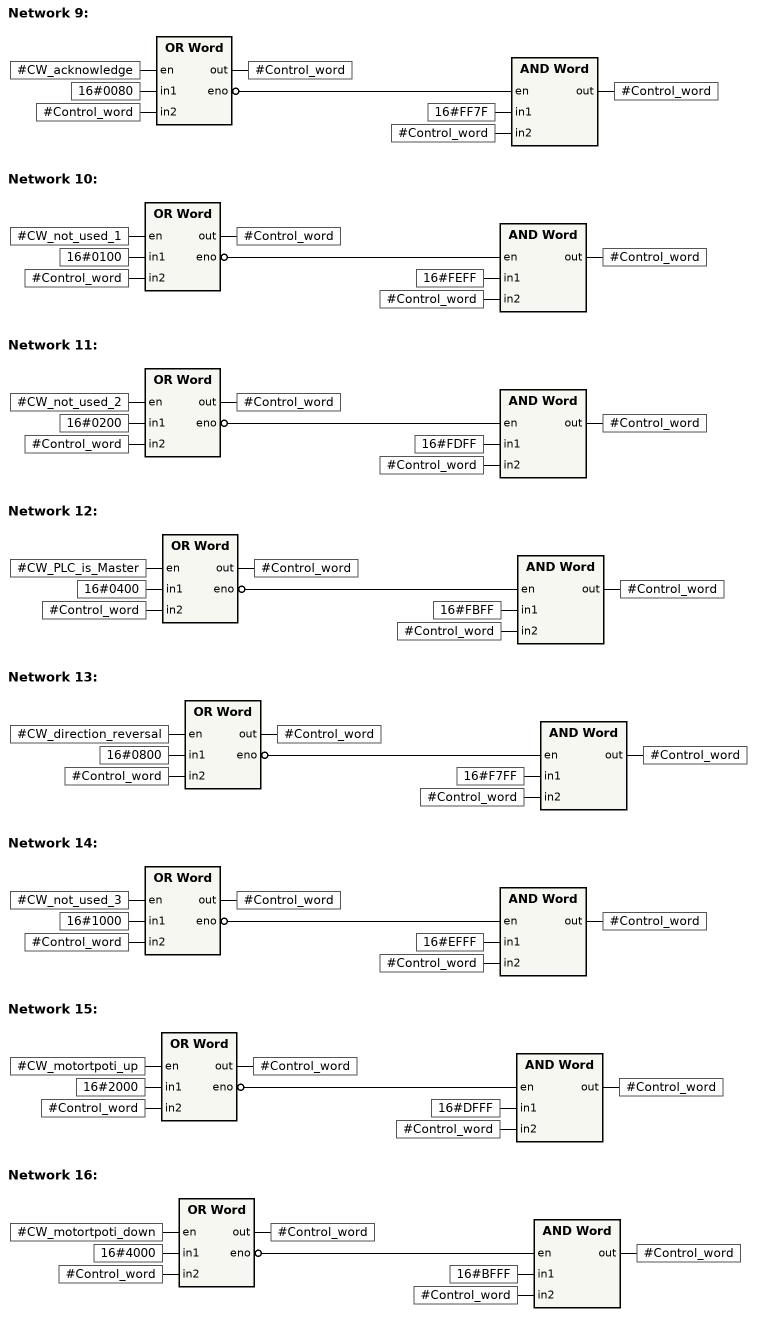
   IF #CW_acknowledge THEN #Control_word := 16#0080 OR #Control_word; END_IF;
   IF NOT #CW_acknowledge THEN #Control_word := 16#FF7F AND #Control_word; END_IF;
END_REGION

REGION Network 10
   IF #CW_not_used_1 THEN #Control_word := 16#0100 OR #Control_word; END_IF;
   IF NOT #CW_not_used_1 THEN #Control_word := 16#FEFF AND #Control_word; END_IF;
END_REGION

REGION Network 11
   IF #CW_not_used_2 THEN #Control_word := 16#0200 OR #Control_word; END_IF;
   IF NOT #CW_not_used_2 THEN #Control_word := 16#FDFF AND #Control_word; END_IF;
END_REGION

REGION Network 12
   IF #CW_PLC_is_Master THEN #Control_word := 16#0400 OR #Control_word; END_IF;
   IF NOT #CW_PLC_is_Master THEN #Control_word := 16#FBFF AND #Control_word; END_IF;
END_REGION

REGION Network 13
   IF #CW_direction_reversal THEN #Control_word := 16#0800 OR #Control_word; END_IF;
   IF NOT #CW_direction_reversal THEN #Control_word := 16#F7FF AND #Control_word; END_IF;
END_REGION

REGION Network 14
   IF #CW_not_used_3 THEN #Control_word := 16#1000 OR #Control_word; END_IF;
   IF NOT #CW_not_used_3 THEN #Control_word := 16#EFFF AND #Control_word; END_IF;
END_REGION

REGION Network 15
   IF #CW_motortpoti_up THEN #Control_word := 16#2000 OR #Control_word; END_IF;
   IF NOT #CW_motortpoti_up THEN #Control_word := 16#DFFF AND #Control_word; END_IF;
END_REGION

REGION Network 16
   IF #CW_motortpoti_down THEN #Control_word := 16#4000 OR #Control_word; END_IF;
   IF NOT #CW_motortpoti_down THEN #Control_word := 16#BFFF AND #Control_word; END_IF;
END_REGION

REGION Network 17
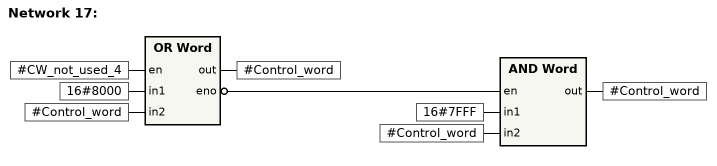
   IF #CW_not_used_4 THEN #Control_word := 16#8000 OR #Control_word; END_IF;
   IF NOT #CW_not_used_4 THEN #Control_word := 16#7FFF AND #Control_word; END_IF;
END_REGION
END_FUNCTION

FUNCTION_BLOCK "Inverter_Process_Data"   // FB1, FBD
{ S7_Optimized_Access := 'TRUE' }
VERSION : 0.1
// stored: AutoNumber false, IsIECCheckEnabled false, IsRetainMemResEnabled false, MemoryReserve 100, SetENOAutomatically false, UDAEnableTagReadback false
   VAR_INPUT
      control_word : Word := 16#0000;
      setpoint : Real;
      RD_address : HW_SUBMODULE;
      WR_address : HW_SUBMODULE;
      ref_quantity : Struct
         speed_p2000 : Real := 1500.0;
         current_p2002 : Real := 0.65;
         torque_p2003 : Real := 1.7;
      END_STRUCT;
   END_VAR
   VAR_OUTPUT
      status_word : Word;
      actual_speed : Real;
      actual_current : Real;
      actual_torque : Real;
      actual_alarm : Word;
      actual_fault : Word;
      RETVAL_RD : Word;
      RETVAL_WR : Word;
   END_VAR
   VAR_TEMP
      InData : Array[1..6] of Word;
      OutData : Array[1..6] of Word;
      actual_speed_INT : Int;
      actual_current_INT : Int;
      actual_torque_INT : Int;
      setpoint_INT : Int;
   END_VAR
BEGIN

REGION Network 1
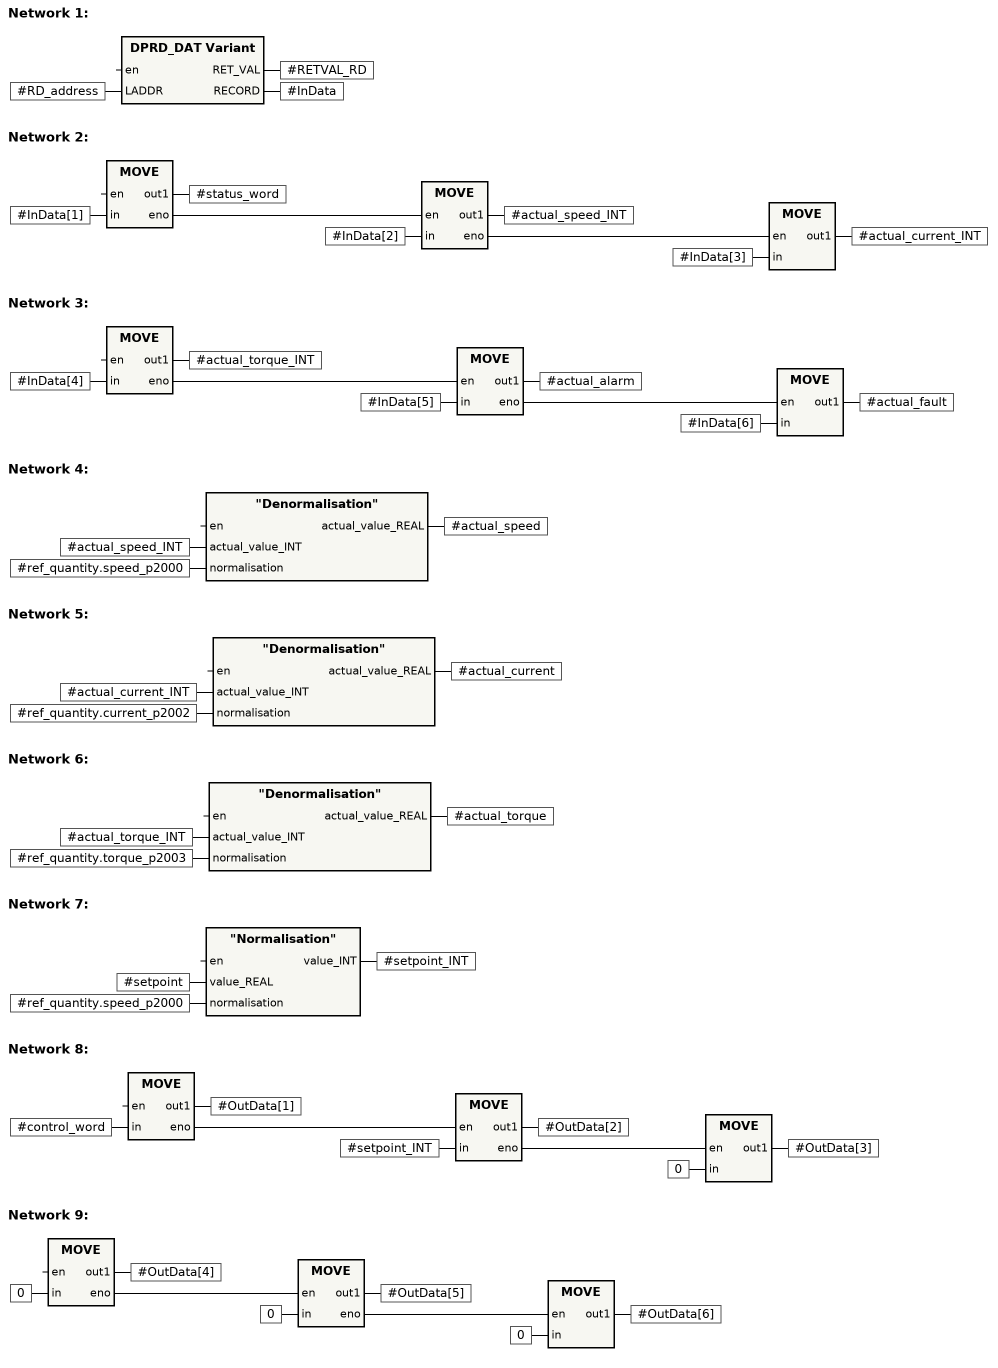
   #RETVAL_RD := DPRD_DAT(LADDR := #RD_address, RECORD => #InData);
END_REGION

REGION Network 2
   // ENO of a box is taken as its EN; it also drops when the box reports an error
   #status_word := #InData[1];
   #actual_speed_INT := #InData[2];
   #actual_current_INT := #InData[3];
END_REGION

REGION Network 3
   // ENO of a box is taken as its EN; it also drops when the box reports an error
   #actual_torque_INT := #InData[4];
   #actual_alarm := #InData[5];
   #actual_fault := #InData[6];
END_REGION

REGION Network 4
   "Denormalisation"(actual_value_INT := #actual_speed_INT,
                     normalisation := #ref_quantity.speed_p2000,
                     actual_value_REAL => #actual_speed);
END_REGION

REGION Network 5
   "Denormalisation"(actual_value_INT := #actual_current_INT,
                     normalisation := #ref_quantity.current_p2002,
                     actual_value_REAL => #actual_current);
END_REGION

REGION Network 6
   "Denormalisation"(actual_value_INT := #actual_torque_INT,
                     normalisation := #ref_quantity.torque_p2003,
                     actual_value_REAL => #actual_torque);
END_REGION

REGION Network 7
   "Normalisation"(value_REAL := #setpoint,
                   normalisation := #ref_quantity.speed_p2000,
                   value_INT => #setpoint_INT);
END_REGION

REGION Network 8
   // ENO of a box is taken as its EN; it also drops when the box reports an error
   #OutData[1] := #control_word;
   #OutData[2] := #setpoint_INT;
   #OutData[3] := 0;
END_REGION

REGION Network 9
   // ENO of a box is taken as its EN; it also drops when the box reports an error
   #OutData[4] := 0;
   #OutData[5] := 0;
   #OutData[6] := 0;
END_REGION

REGION Network 10
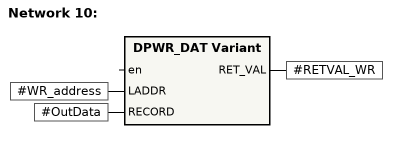
   #RETVAL_WR := DPWR_DAT(LADDR := #WR_address, RECORD := #OutData);
END_REGION
END_FUNCTION_BLOCK

FUNCTION_BLOCK "Modbus"   // FB20, FBD
{ S7_Optimized_Access := 'FALSE' }
VERSION : 0.1
// stored: AutoNumber false, IsIECCheckEnabled false, SetENOAutomatically false, UDAEnableTagReadback false
   VAR_INPUT
      BAUDRATE : UDInt := 115200;
      HW_ID : PORT := 272;
      RESP_TO : UInt := 1000;
      CYCLIC_PROCESSING : Bool := true;
      MB_ADDR : UInt := 8;
      DATA_AD_R : UDInt := 40001;
      DATA_AD_W : UDInt := 40006;
      DATA_LEN_R : UInt := 5;
      DATA_LEN_W : UInt := 5;
      ReadOnly : Bool := 1;   // Read only (1)
   END_VAR
   VAR_OUTPUT
      ERROR : Bool;
      ERROR_INFO : Struct
         drive_number : USInt;
         "step" : USInt;
         STATUS : Word;
      END_STRUCT;
   END_VAR
   VAR_IN_OUT
      ReadDone_0 : Bool;   // Read done for prestretch board (1)
      DT_PTR_IN : Variant;
      DT_PTR_OUT : Variant;
   END_VAR
   VAR DB_SPECIFIC
      drive_index : USInt := 1;
      "step" : USInt := 0;
      REQ : Bool;
      extended_restart : Bool;
      start_internal : Bool;
   END_VAR
   VAR
      MB_COMM_LOAD_Instance { S7_SetPoint := 'True'} : MB_COMM_LOAD;
      MB_MASTER_Instance { S7_SetPoint := 'True'} : MB_MASTER;
   END_VAR
   VAR_TEMP
      _DONE : Bool;
      _ERROR : Bool;
      _STATUS : Word;
      _cyclic_processing : Bool;
   END_VAR
   VAR_TEMP   // added for the SCL form of the ladder/FBD networks
      _w1 : Bool;
      _w2 : Bool;
      _w3 : Bool;
   END_VAR
BEGIN

REGION Network 1: First cycle
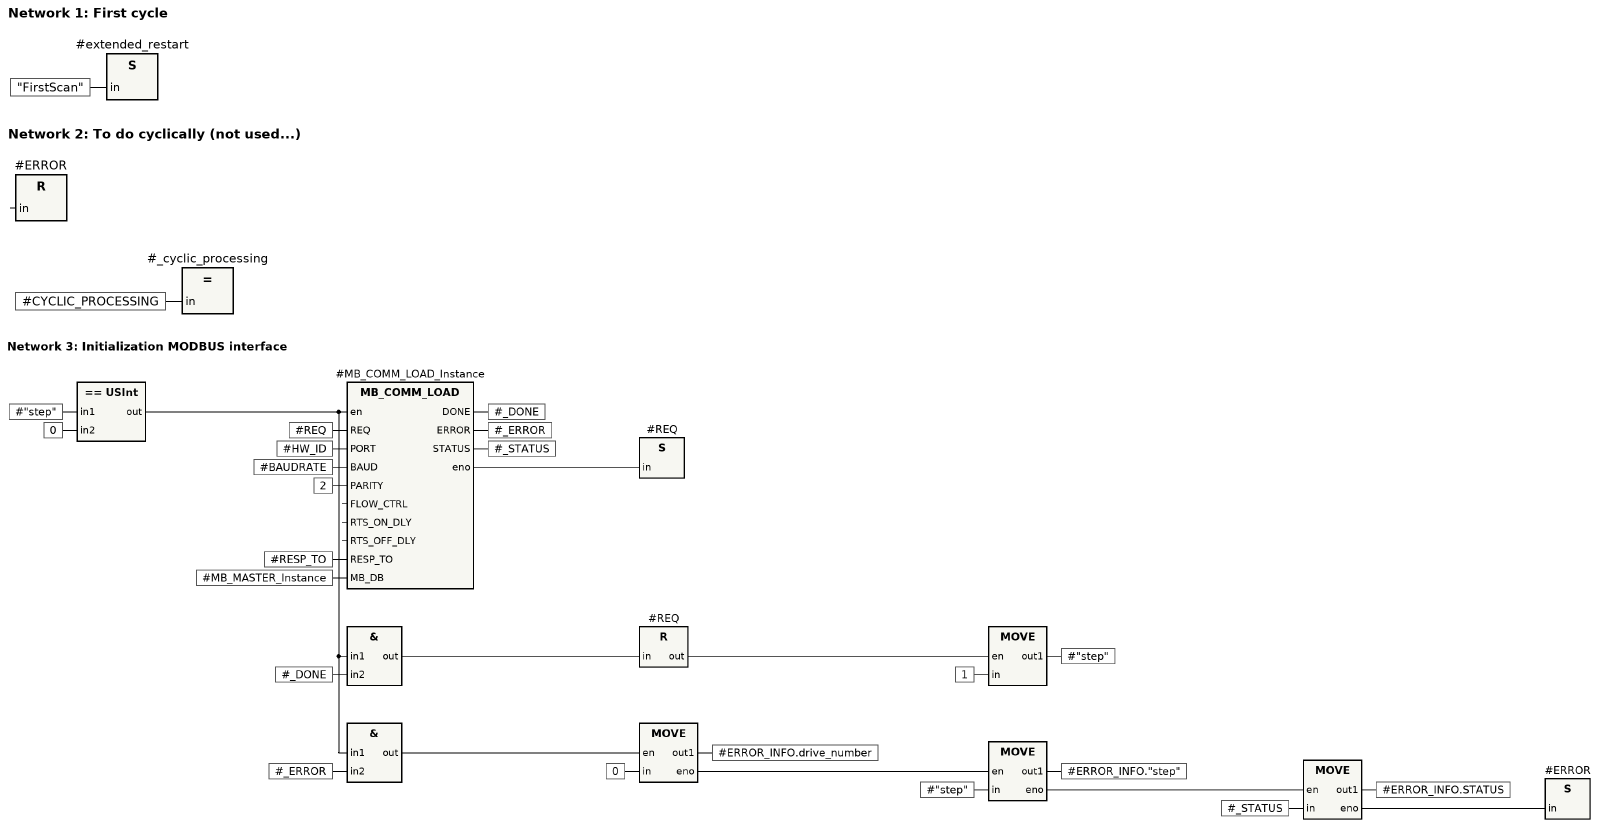
   IF "FirstScan" THEN #extended_restart := TRUE; END_IF;
END_REGION

REGION Network 2: To do cyclically (not used...)
   #ERROR := FALSE;
   #_cyclic_processing := #CYCLIC_PROCESSING;
END_REGION

REGION Network 3: Initialization MODBUS interface
   // ENO of a box is taken as its EN; it also drops when the box reports an error
   #_w1 := #"step" = 0;
   #MB_COMM_LOAD_Instance(EN := #_w1,   // MB_COMM_LOAD
                          REQ := #REQ,
                          PORT := #HW_ID,
                          BAUD := #BAUDRATE,
                          PARITY := 2,
                          RESP_TO := #RESP_TO,
                          MB_DB := #MB_MASTER_Instance,
                          DONE => #_DONE,
                          ERROR => #_ERROR,
                          STATUS => #_STATUS,
                          ENO => #_w2);
   IF #_w2 THEN #REQ := TRUE; END_IF;
   IF #_w1 AND #_DONE THEN
       #REQ := FALSE;
       #"step" := 1;
   END_IF;
   IF #_w1 AND #_ERROR THEN
       #ERROR_INFO.drive_number := 0;
       #ERROR_INFO."step" := #"step";
       #ERROR_INFO.STATUS := #_STATUS;
       #ERROR := TRUE;
   END_IF;
END_REGION

REGION Network 4: READ
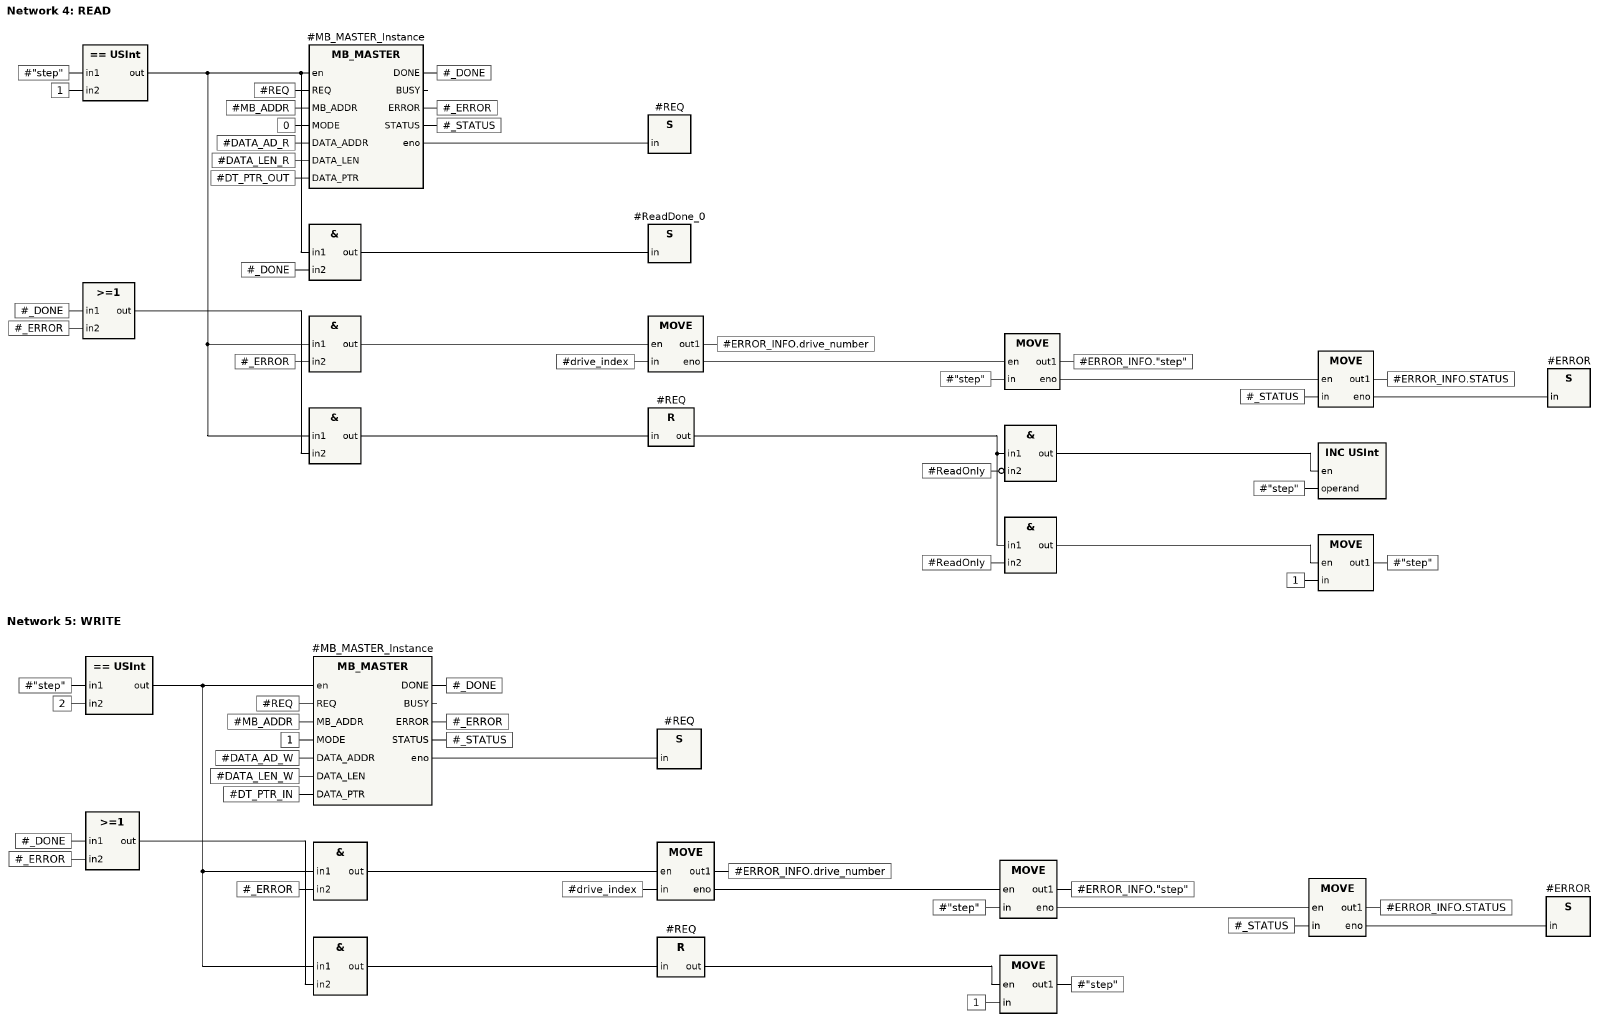
   // ENO of a box is taken as its EN; it also drops when the box reports an error
   #_w1 := #"step" = 1;
   #MB_MASTER_Instance(EN := #_w1,   // MB_MASTER
                       REQ := #REQ,
                       MB_ADDR := #MB_ADDR,
                       MODE := 0,
                       DATA_ADDR := #DATA_AD_R,
                       DATA_LEN := #DATA_LEN_R,
                       DATA_PTR := #DT_PTR_OUT,
                       DONE => #_DONE,
                       ERROR => #_ERROR,
                       STATUS => #_STATUS,
                       ENO => #_w2);
   IF #_w2 THEN #REQ := TRUE; END_IF;
   IF #_w1 AND #_DONE THEN #ReadDone_0 := TRUE; END_IF;
   IF #_w1 AND #_ERROR THEN
       #ERROR_INFO.drive_number := #drive_index;
       #ERROR_INFO."step" := #"step";
       #ERROR_INFO.STATUS := #_STATUS;
       #ERROR := TRUE;
   END_IF;
   #_w3 := #_w1 AND (#_DONE OR #_ERROR);
   IF #_w3 THEN #REQ := FALSE; END_IF;
   IF #_w3 AND NOT #ReadOnly THEN #"step" := #"step" + 1; END_IF;
   IF #_w3 AND #ReadOnly THEN #"step" := 1; END_IF;
END_REGION

REGION Network 5: WRITE
   // ENO of a box is taken as its EN; it also drops when the box reports an error
   #_w1 := #"step" = 2;
   #MB_MASTER_Instance(EN := #_w1,   // MB_MASTER
                       REQ := #REQ,
                       MB_ADDR := #MB_ADDR,
                       MODE := 1,
                       DATA_ADDR := #DATA_AD_W,
                       DATA_LEN := #DATA_LEN_W,
                       DATA_PTR := #DT_PTR_IN,
                       DONE => #_DONE,
                       ERROR => #_ERROR,
                       STATUS => #_STATUS,
                       ENO => #_w2);
   IF #_w2 THEN #REQ := TRUE; END_IF;
   IF #_w1 AND #_ERROR THEN
       #ERROR_INFO.drive_number := #drive_index;
       #ERROR_INFO."step" := #"step";
       #ERROR_INFO.STATUS := #_STATUS;
       #ERROR := TRUE;
   END_IF;
   IF #_w1 AND (#_DONE OR #_ERROR) THEN
       #REQ := FALSE;
       #"step" := 1;
   END_IF;
END_REGION
END_FUNCTION_BLOCK

FUNCTION "Proc_Analog_Press_Filt1" : Void   // FC18, LAD
{ S7_Optimized_Access := 'TRUE' }
VERSION : 0.1
// stored: AutoNumber true, IsIECCheckEnabled false, SetENOAutomatically false, UDAEnableTagReadback false
   VAR_OUTPUT
      Pressão_em_Bar : Real;
   END_VAR
   VAR_TEMP
      "Pressão_em_%" : Real;
   END_VAR
BEGIN

REGION Network 1
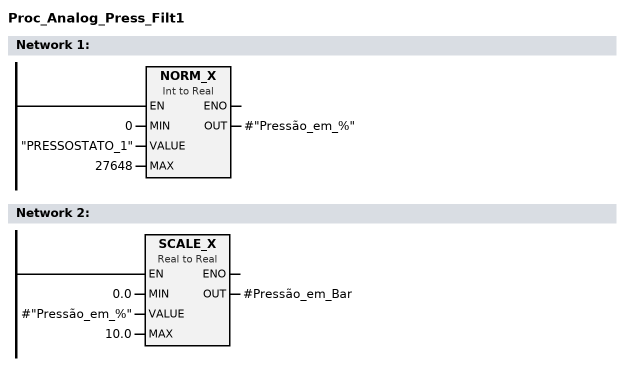
   RUNG wire#powerrail
      { S7_Templates := "[SrcType := Int, DestType := Real]"; S7_GenerateENO := "TRUE" } Normalize(min := 0, value := "PRESSOSTATO_1", max := 27648, out => #"Pressão_em_%")
   END_RUNG
   // the same network as SCL:
   #"Pressão_em_%" := NORM_X(MIN := 0, VALUE := "PRESSOSTATO_1", MAX := 27648);
END_REGION

REGION Network 2
   RUNG wire#powerrail
      { S7_Templates := "[SrcType := Real, DestType := Real]"; S7_GenerateENO := "TRUE" } Scale(min := 0.0, value := #"Pressão_em_%", max := 10.0, out => #Pressão_em_Bar)
   END_RUNG
   // the same network as SCL:
   #Pressão_em_Bar := SCALE_X(MIN := 0.0, VALUE := #"Pressão_em_%", MAX := 10.0);
END_REGION
END_FUNCTION

FUNCTION "Proc_Analog_Press_Filt2" : Void   // FC19, LAD
{ S7_Optimized_Access := 'TRUE' }
VERSION : 0.1
// stored: AutoNumber true, IsIECCheckEnabled false, SetENOAutomatically false, UDAEnableTagReadback false
   VAR_OUTPUT
      Pressão_em_Bar : Real;
   END_VAR
   VAR_TEMP
      "Pressão_em_%" : Real;
   END_VAR
BEGIN

REGION Network 1
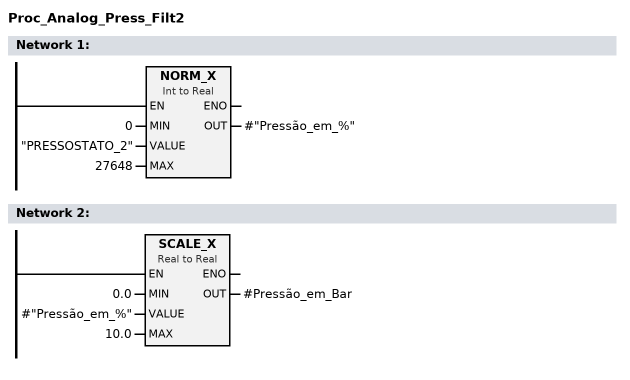
   RUNG wire#powerrail
      { S7_Templates := "[SrcType := Int, DestType := Real]"; S7_GenerateENO := "TRUE" } Normalize(min := 0, value := "PRESSOSTATO_2", max := 27648, out => #"Pressão_em_%")
   END_RUNG
   // the same network as SCL:
   #"Pressão_em_%" := NORM_X(MIN := 0, VALUE := "PRESSOSTATO_2", MAX := 27648);
END_REGION

REGION Network 2
   RUNG wire#powerrail
      { S7_Templates := "[SrcType := Real, DestType := Real]"; S7_GenerateENO := "TRUE" } Scale(min := 0.0, value := #"Pressão_em_%", max := 10.0, out => #Pressão_em_Bar)
   END_RUNG
   // the same network as SCL:
   #Pressão_em_Bar := SCALE_X(MIN := 0.0, VALUE := #"Pressão_em_%", MAX := 10.0);
END_REGION
END_FUNCTION

FUNCTION "Saídas_Bombas_Temporário" : Void   // FC17, LAD
{ S7_Optimized_Access := 'TRUE' }
VERSION : 0.1
// stored: AutoNumber true, IsIECCheckEnabled false, SetENOAutomatically false, UDAEnableTagReadback false
BEGIN

REGION Network 1
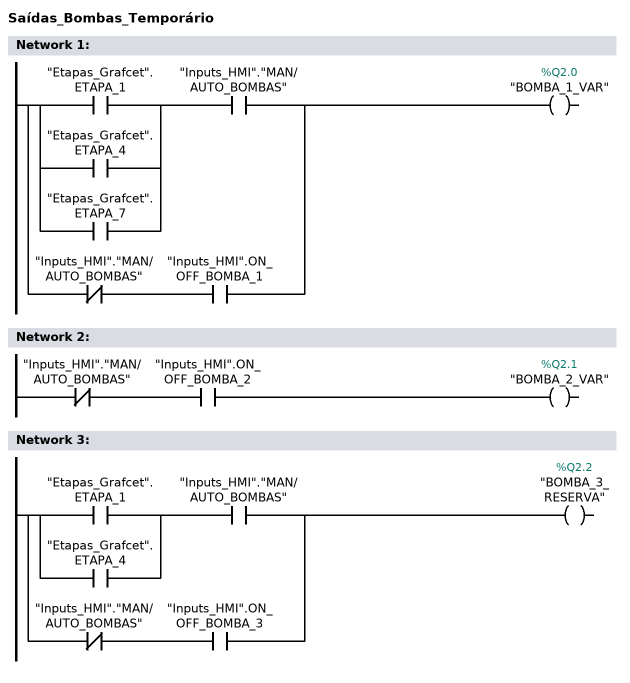
   RUNG wire#powerrail
      Contact( "Etapas_Grafcet".ETAPA_1 )
      wire#w1
      Contact( "Inputs_HMI"."MAN/AUTO_BOMBAS" )
      wire#w2
      Coil( "BOMBA_1_VAR" )
   END_RUNG
   RUNG wire#powerrail
      Contact( "Etapas_Grafcet".ETAPA_4 )
   END_RUNG wire#w1
   RUNG wire#powerrail
      Contact( "Etapas_Grafcet".ETAPA_7 )
   END_RUNG wire#w1
   RUNG wire#powerrail
      I_Contact( "Inputs_HMI"."MAN/AUTO_BOMBAS" )
      Contact( "Inputs_HMI".ON_OFF_BOMBA_1 )
   END_RUNG wire#w2
   // the same network as SCL:
   "BOMBA_1_VAR" := (("Etapas_Grafcet".ETAPA_1 OR "Etapas_Grafcet".ETAPA_4 OR "Etapas_Grafcet".ETAPA_7) AND "Inputs_HMI"."MAN/AUTO_BOMBAS") OR (NOT "Inputs_HMI"."MAN/AUTO_BOMBAS" AND "Inputs_HMI".ON_OFF_BOMBA_1);
END_REGION

REGION Network 2
   RUNG wire#powerrail
      I_Contact( "Inputs_HMI"."MAN/AUTO_BOMBAS" )
      Contact( "Inputs_HMI".ON_OFF_BOMBA_2 )
      Coil( "BOMBA_2_VAR" )
   END_RUNG
   // the same network as SCL:
   "BOMBA_2_VAR" := NOT "Inputs_HMI"."MAN/AUTO_BOMBAS" AND "Inputs_HMI".ON_OFF_BOMBA_2;
END_REGION

REGION Network 3
   RUNG wire#powerrail
      Contact( "Etapas_Grafcet".ETAPA_1 )
      wire#w1
      Contact( "Inputs_HMI"."MAN/AUTO_BOMBAS" )
      wire#w2
      Coil( "BOMBA_3_RESERVA" )
   END_RUNG
   RUNG wire#powerrail
      Contact( "Etapas_Grafcet".ETAPA_4 )
   END_RUNG wire#w1
   RUNG wire#powerrail
      I_Contact( "Inputs_HMI"."MAN/AUTO_BOMBAS" )
      Contact( "Inputs_HMI".ON_OFF_BOMBA_3 )
   END_RUNG wire#w2
   // the same network as SCL:
   "BOMBA_3_RESERVA" := (("Etapas_Grafcet".ETAPA_1 OR "Etapas_Grafcet".ETAPA_4) AND "Inputs_HMI"."MAN/AUTO_BOMBAS") OR (NOT "Inputs_HMI"."MAN/AUTO_BOMBAS" AND "Inputs_HMI".ON_OFF_BOMBA_3);
END_REGION
END_FUNCTION

FUNCTION "Alarme_XV102" : Void   // FC24, LAD
{ S7_Optimized_Access := 'TRUE' }
VERSION : 0.1
// stored: AutoNumber true, IsIECCheckEnabled false, SetENOAutomatically false, UDAEnableTagReadback false
BEGIN

REGION Network 1: XV102 a abrir
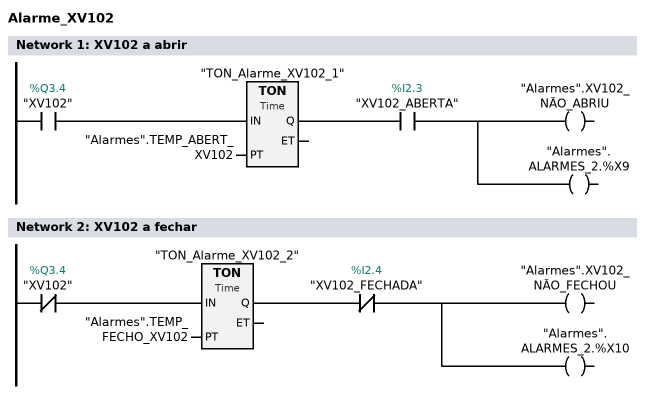
   RUNG wire#powerrail
      Contact( "XV102" )
      { S7_Templates := "time_type := Time" } "TON_Alarme_XV102_1".TON(pt := "Alarmes".TEMP_ABERT_XV102, et =>)
      Contact( "XV102_ABERTA" )
      wire#w1
      Coil( "Alarmes".XV102_NÃO_ABRIU )
   END_RUNG
   RUNG wire#w1
      Coil( "Alarmes".ALARMES_2.%X9 )
   END_RUNG
   // the same network as SCL:
   "TON_Alarme_XV102_1".TON(IN := "XV102", PT := "Alarmes".TEMP_ABERT_XV102);
   "Alarmes".XV102_NÃO_ABRIU := "TON_Alarme_XV102_1".Q AND "XV102_ABERTA";
   "Alarmes".ALARMES_2.%X9 := "Alarmes".XV102_NÃO_ABRIU;
END_REGION

REGION Network 2: XV102 a fechar
   RUNG wire#powerrail
      I_Contact( "XV102" )
      { S7_Templates := "time_type := Time" } "TON_Alarme_XV102_2".TON(pt := "Alarmes".TEMP_FECHO_XV102, et =>)
      I_Contact( "XV102_FECHADA" )
      wire#w1
      Coil( "Alarmes".XV102_NÃO_FECHOU )
   END_RUNG
   RUNG wire#w1
      Coil( "Alarmes".ALARMES_2.%X10 )
   END_RUNG
   // the same network as SCL:
   "TON_Alarme_XV102_2".TON(IN := NOT "XV102", PT := "Alarmes".TEMP_FECHO_XV102);
   "Alarmes".XV102_NÃO_FECHOU := "TON_Alarme_XV102_2".Q AND NOT "XV102_FECHADA";
   "Alarmes".ALARMES_2.%X10 := "Alarmes".XV102_NÃO_FECHOU;
END_REGION
END_FUNCTION

FUNCTION "Alarmes_Disparos_1" : Void   // FC22, LAD
{ S7_Optimized_Access := 'TRUE' }
VERSION : 0.1
// stored: AutoNumber true, IsIECCheckEnabled false, SetENOAutomatically false, UDAEnableTagReadback false
   VAR_TEMP   // added for the SCL form of the ladder/FBD networks
      _w1 : Bool;
      _w2 : Bool;
      _w3 : Bool;
      _w4 : Bool;
      _w5 : Bool;
      _w6 : Bool;
      _w7 : Bool;
      _w8 : Bool;
      _w9 : Bool;
      _w10 : Bool;
      _w11 : Bool;
      _w12 : Bool;
      _w13 : Bool;
      _w14 : Bool;
      _w15 : Bool;
      _w16 : Bool;
      _w17 : Bool;
      _w18 : Bool;
      _w19 : Bool;
      _w20 : Bool;
      _w21 : Bool;
      _w22 : Bool;
   END_VAR
BEGIN

REGION Network 1: Ativa contacto de alarme disparos para alarme luminoso
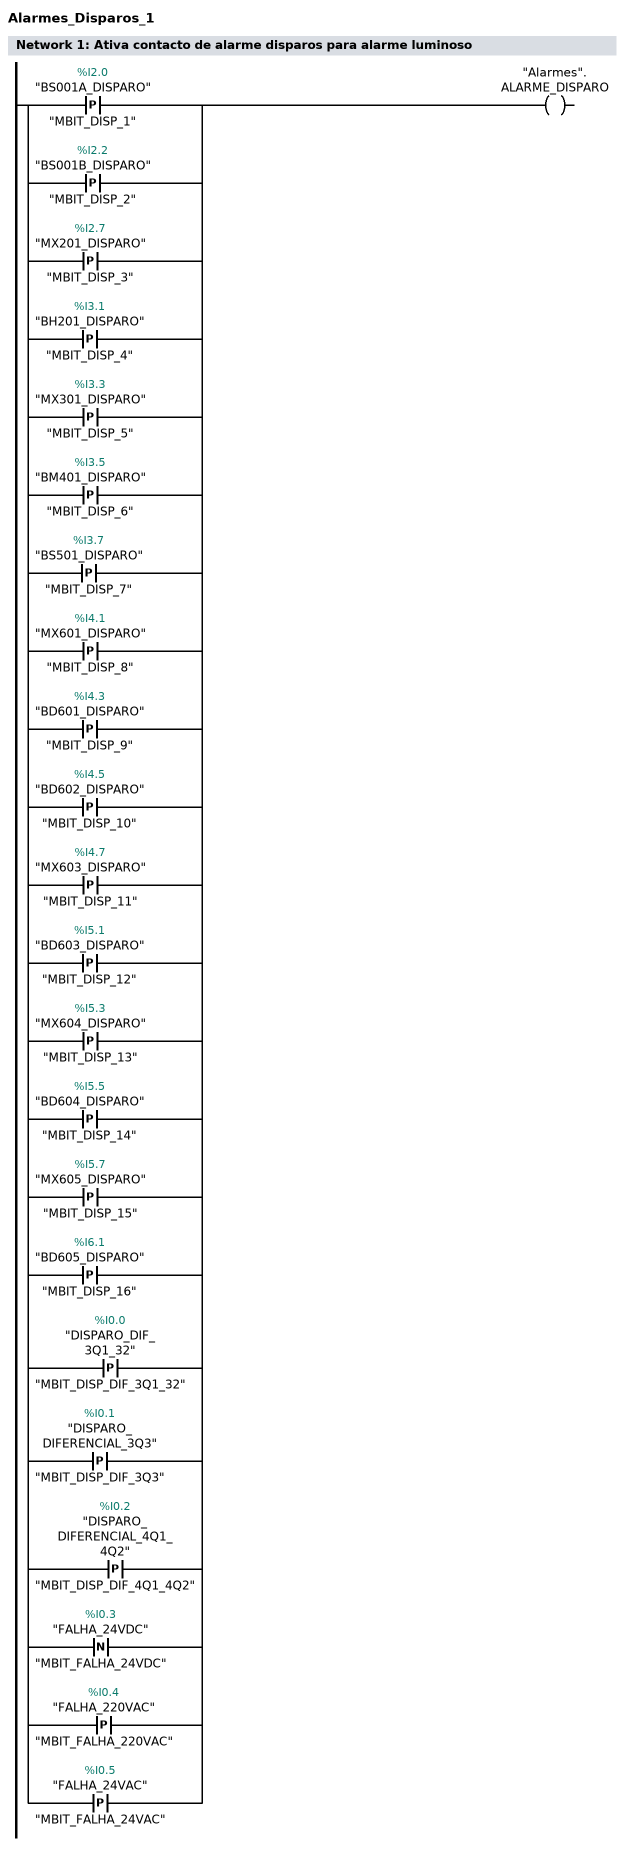
   RUNG wire#powerrail
      P_Contact(operand := "BS001A_DISPARO", bit := "MBIT_DISP_1")
      wire#w1
      Coil( "Alarmes".ALARME_DISPARO )
   END_RUNG
   RUNG wire#powerrail
      P_Contact(operand := "BS001B_DISPARO", bit := "MBIT_DISP_2")
   END_RUNG wire#w1
   RUNG wire#powerrail
      P_Contact(operand := "MX201_DISPARO", bit := "MBIT_DISP_3")
   END_RUNG wire#w1
   RUNG wire#powerrail
      P_Contact(operand := "BH201_DISPARO", bit := "MBIT_DISP_4")
   END_RUNG wire#w1
   RUNG wire#powerrail
      P_Contact(operand := "MX301_DISPARO", bit := "MBIT_DISP_5")
   END_RUNG wire#w1
   RUNG wire#powerrail
      P_Contact(operand := "BM401_DISPARO", bit := "MBIT_DISP_6")
   END_RUNG wire#w1
   RUNG wire#powerrail
      P_Contact(operand := "BS501_DISPARO", bit := "MBIT_DISP_7")
   END_RUNG wire#w1
   RUNG wire#powerrail
      P_Contact(operand := "MX601_DISPARO", bit := "MBIT_DISP_8")
   END_RUNG wire#w1
   RUNG wire#powerrail
      P_Contact(operand := "BD601_DISPARO", bit := "MBIT_DISP_9")
   END_RUNG wire#w1
   RUNG wire#powerrail
      P_Contact(operand := "BD602_DISPARO", bit := "MBIT_DISP_10")
   END_RUNG wire#w1
   RUNG wire#powerrail
      P_Contact(operand := "MX603_DISPARO", bit := "MBIT_DISP_11")
   END_RUNG wire#w1
   RUNG wire#powerrail
      P_Contact(operand := "BD603_DISPARO", bit := "MBIT_DISP_12")
   END_RUNG wire#w1
   RUNG wire#powerrail
      P_Contact(operand := "MX604_DISPARO", bit := "MBIT_DISP_13")
   END_RUNG wire#w1
   RUNG wire#powerrail
      P_Contact(operand := "BD604_DISPARO", bit := "MBIT_DISP_14")
   END_RUNG wire#w1
   RUNG wire#powerrail
      P_Contact(operand := "MX605_DISPARO", bit := "MBIT_DISP_15")
   END_RUNG wire#w1
   RUNG wire#powerrail
      P_Contact(operand := "BD605_DISPARO", bit := "MBIT_DISP_16")
   END_RUNG wire#w1
   RUNG wire#powerrail
      P_Contact(operand := "DISPARO_DIF_3Q1_32", bit := "MBIT_DISP_DIF_3Q1_32")
   END_RUNG wire#w1
   RUNG wire#powerrail
      P_Contact(operand := "DISPARO_DIFERENCIAL_3Q3", bit := "MBIT_DISP_DIF_3Q3")
   END_RUNG wire#w1
   RUNG wire#powerrail
      P_Contact(operand := "DISPARO_DIFERENCIAL_4Q1_4Q2", bit := "MBIT_DISP_DIF_4Q1_4Q2")
   END_RUNG wire#w1
   RUNG wire#powerrail
      N_Contact(operand := "FALHA_24VDC", bit := "MBIT_FALHA_24VDC")
   END_RUNG wire#w1
   RUNG wire#powerrail
      P_Contact(operand := "FALHA_220VAC", bit := "MBIT_FALHA_220VAC")
   END_RUNG wire#w1
   RUNG wire#powerrail
      P_Contact(operand := "FALHA_24VAC", bit := "MBIT_FALHA_24VAC")
   END_RUNG wire#w1
   // the same network as SCL:
   #_w1 := "BS001A_DISPARO" AND NOT "MBIT_DISP_1";   // rising edge of "BS001A_DISPARO"
   "MBIT_DISP_1" := "BS001A_DISPARO";
   #_w2 := "BS001B_DISPARO" AND NOT "MBIT_DISP_2";   // rising edge of "BS001B_DISPARO"
   "MBIT_DISP_2" := "BS001B_DISPARO";
   #_w3 := "MX201_DISPARO" AND NOT "MBIT_DISP_3";   // rising edge of "MX201_DISPARO"
   "MBIT_DISP_3" := "MX201_DISPARO";
   #_w4 := "BH201_DISPARO" AND NOT "MBIT_DISP_4";   // rising edge of "BH201_DISPARO"
   "MBIT_DISP_4" := "BH201_DISPARO";
   #_w5 := "MX301_DISPARO" AND NOT "MBIT_DISP_5";   // rising edge of "MX301_DISPARO"
   "MBIT_DISP_5" := "MX301_DISPARO";
   #_w6 := "BM401_DISPARO" AND NOT "MBIT_DISP_6";   // rising edge of "BM401_DISPARO"
   "MBIT_DISP_6" := "BM401_DISPARO";
   #_w7 := "BS501_DISPARO" AND NOT "MBIT_DISP_7";   // rising edge of "BS501_DISPARO"
   "MBIT_DISP_7" := "BS501_DISPARO";
   #_w8 := "MX601_DISPARO" AND NOT "MBIT_DISP_8";   // rising edge of "MX601_DISPARO"
   "MBIT_DISP_8" := "MX601_DISPARO";
   #_w9 := "BD601_DISPARO" AND NOT "MBIT_DISP_9";   // rising edge of "BD601_DISPARO"
   "MBIT_DISP_9" := "BD601_DISPARO";
   #_w10 := "BD602_DISPARO" AND NOT "MBIT_DISP_10";   // rising edge of "BD602_DISPARO"
   "MBIT_DISP_10" := "BD602_DISPARO";
   #_w11 := "MX603_DISPARO" AND NOT "MBIT_DISP_11";   // rising edge of "MX603_DISPARO"
   "MBIT_DISP_11" := "MX603_DISPARO";
   #_w12 := "BD603_DISPARO" AND NOT "MBIT_DISP_12";   // rising edge of "BD603_DISPARO"
   "MBIT_DISP_12" := "BD603_DISPARO";
   #_w13 := "MX604_DISPARO" AND NOT "MBIT_DISP_13";   // rising edge of "MX604_DISPARO"
   "MBIT_DISP_13" := "MX604_DISPARO";
   #_w14 := "BD604_DISPARO" AND NOT "MBIT_DISP_14";   // rising edge of "BD604_DISPARO"
   "MBIT_DISP_14" := "BD604_DISPARO";
   #_w15 := "MX605_DISPARO" AND NOT "MBIT_DISP_15";   // rising edge of "MX605_DISPARO"
   "MBIT_DISP_15" := "MX605_DISPARO";
   #_w16 := "BD605_DISPARO" AND NOT "MBIT_DISP_16";   // rising edge of "BD605_DISPARO"
   "MBIT_DISP_16" := "BD605_DISPARO";
   #_w17 := "DISPARO_DIF_3Q1_32" AND NOT "MBIT_DISP_DIF_3Q1_32";   // rising edge of "DISPARO_DIF_3Q1_32"
   "MBIT_DISP_DIF_3Q1_32" := "DISPARO_DIF_3Q1_32";
   #_w18 := "DISPARO_DIFERENCIAL_3Q3" AND NOT "MBIT_DISP_DIF_3Q3";   // rising edge of "DISPARO_DIFERENCIAL_3Q3"
   "MBIT_DISP_DIF_3Q3" := "DISPARO_DIFERENCIAL_3Q3";
   #_w19 := "DISPARO_DIFERENCIAL_4Q1_4Q2" AND NOT "MBIT_DISP_DIF_4Q1_4Q2";   // rising edge of "DISPARO_DIFERENCIAL_4Q1_4Q2"
   "MBIT_DISP_DIF_4Q1_4Q2" := "DISPARO_DIFERENCIAL_4Q1_4Q2";
   #_w20 := NOT "FALHA_24VDC" AND "MBIT_FALHA_24VDC";   // falling edge of "FALHA_24VDC"
   "MBIT_FALHA_24VDC" := "FALHA_24VDC";
   #_w21 := "FALHA_220VAC" AND NOT "MBIT_FALHA_220VAC";   // rising edge of "FALHA_220VAC"
   "MBIT_FALHA_220VAC" := "FALHA_220VAC";
   #_w22 := "FALHA_24VAC" AND NOT "MBIT_FALHA_24VAC";   // rising edge of "FALHA_24VAC"
   "MBIT_FALHA_24VAC" := "FALHA_24VAC";
   "Alarmes".ALARME_DISPARO := #_w1 OR #_w2 OR #_w3 OR #_w4 OR #_w5 OR #_w6 OR #_w7 OR #_w8 OR #_w9 OR #_w10 OR #_w11 OR #_w12 OR #_w13 OR #_w14 OR #_w15 OR #_w16 OR #_w17 OR #_w18 OR #_w19 OR #_w20 OR #_w21 OR #_w22;
END_REGION
END_FUNCTION

FUNCTION "Contador_de_Ciclos" : Void   // FC21, LAD
{ S7_Optimized_Access := 'TRUE' }
VERSION : 0.1
// stored: AutoNumber true, IsIECCheckEnabled false, SetENOAutomatically false, UDAEnableTagReadback false
BEGIN

REGION Network 1: Conta o número de ciclos de tratamento
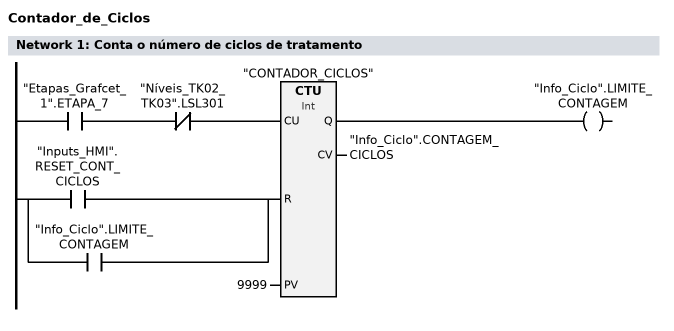
   RUNG wire#powerrail
      Contact( "Etapas_Grafcet_1".ETAPA_7 )
      I_Contact( "Níveis_TK02_TK03".LSL301 )
      { S7_Templates := "value_type := Int" } "CONTADOR_CICLOS".CTU(r := wire#w1, pv := 9999, cv => "Info_Ciclo".CONTAGEM_CICLOS)
      Coil( "Info_Ciclo".LIMITE_CONTAGEM )
   END_RUNG
   RUNG wire#powerrail
      Contact( "Inputs_HMI".RESET_CONT_CICLOS )
   END_RUNG wire#w1
   RUNG wire#powerrail
      Contact( "Info_Ciclo".LIMITE_CONTAGEM )
   END_RUNG wire#w1
   // the same network as SCL:
   "CONTADOR_CICLOS".CTU(CU := "Etapas_Grafcet_1".ETAPA_7 AND NOT "Níveis_TK02_TK03".LSL301,
                         R := "Inputs_HMI".RESET_CONT_CICLOS OR "Info_Ciclo".LIMITE_CONTAGEM,
                         PV := 9999,
                         CV => "Info_Ciclo".CONTAGEM_CICLOS);
   "Info_Ciclo".LIMITE_CONTAGEM := "CONTADOR_CICLOS".Q;
END_REGION
END_FUNCTION

FUNCTION "Reinício_Ciclo" : Void   // FC19, LAD
{ S7_Optimized_Access := 'TRUE' }
VERSION : 0.1
// stored: AutoNumber true, IsIECCheckEnabled false, SetENOAutomatically false, UDAEnableTagReadback false
   VAR_TEMP   // added for the SCL form of the ladder/FBD networks
      _w1 : Bool;
   END_VAR
BEGIN

REGION Network 1: Ativa etapa 1 e faz reset às restantes do ciclo de tratamento
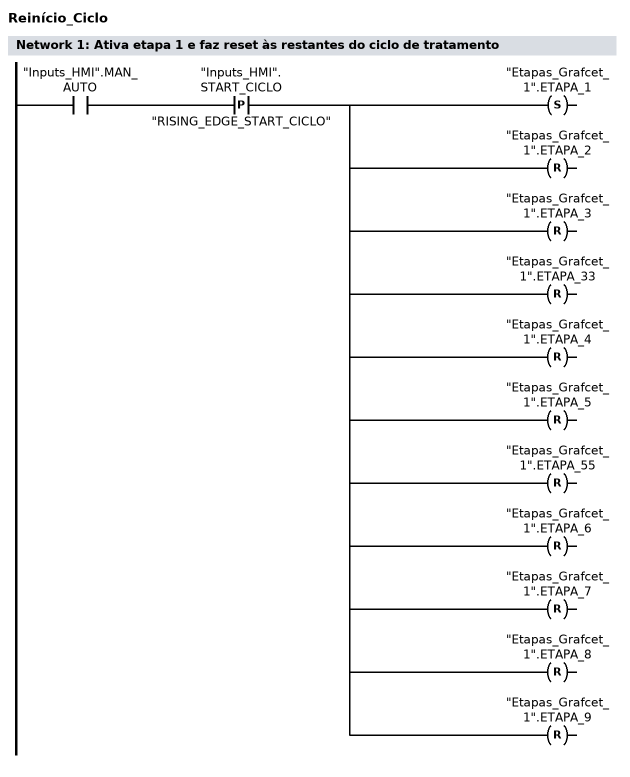
   RUNG wire#powerrail
      Contact( "Inputs_HMI".MAN_AUTO )
      P_Contact(operand := "Inputs_HMI".START_CICLO, bit := "RISING_EDGE_START_CICLO")
      wire#w1
      S_Coil( "Etapas_Grafcet_1".ETAPA_1 )
   END_RUNG
   RUNG wire#w1
      R_Coil( "Etapas_Grafcet_1".ETAPA_2 )
   END_RUNG
   RUNG wire#w1
      R_Coil( "Etapas_Grafcet_1".ETAPA_3 )
   END_RUNG
   RUNG wire#w1
      R_Coil( "Etapas_Grafcet_1".ETAPA_33 )
   END_RUNG
   RUNG wire#w1
      R_Coil( "Etapas_Grafcet_1".ETAPA_4 )
   END_RUNG
   RUNG wire#w1
      R_Coil( "Etapas_Grafcet_1".ETAPA_5 )
   END_RUNG
   RUNG wire#w1
      R_Coil( "Etapas_Grafcet_1".ETAPA_55 )
   END_RUNG
   RUNG wire#w1
      R_Coil( "Etapas_Grafcet_1".ETAPA_6 )
   END_RUNG
   RUNG wire#w1
      R_Coil( "Etapas_Grafcet_1".ETAPA_7 )
   END_RUNG
   RUNG wire#w1
      R_Coil( "Etapas_Grafcet_1".ETAPA_8 )
   END_RUNG
   RUNG wire#w1
      R_Coil( "Etapas_Grafcet_1".ETAPA_9 )
   END_RUNG
   // the same network as SCL:
   #_w1 := "Inputs_HMI".MAN_AUTO AND "Inputs_HMI".START_CICLO AND NOT "RISING_EDGE_START_CICLO";   // rising edge of "Inputs_HMI".START_CICLO
   "RISING_EDGE_START_CICLO" := "Inputs_HMI".START_CICLO;
   IF #_w1 THEN
       "Etapas_Grafcet_1".ETAPA_1 := TRUE;
       "Etapas_Grafcet_1".ETAPA_2 := FALSE;
       "Etapas_Grafcet_1".ETAPA_3 := FALSE;
       "Etapas_Grafcet_1".ETAPA_33 := FALSE;
       "Etapas_Grafcet_1".ETAPA_4 := FALSE;
       "Etapas_Grafcet_1".ETAPA_5 := FALSE;
       "Etapas_Grafcet_1".ETAPA_55 := FALSE;
       "Etapas_Grafcet_1".ETAPA_6 := FALSE;
       "Etapas_Grafcet_1".ETAPA_7 := FALSE;
       "Etapas_Grafcet_1".ETAPA_8 := FALSE;
       "Etapas_Grafcet_1".ETAPA_9 := FALSE;
   END_IF;
END_REGION
END_FUNCTION

FUNCTION "Medidor_Caudal_FQ301" : Void   // FC11, LAD
{ S7_Optimized_Access := 'TRUE' }
VERSION : 0.1
// stored: AutoNumber true, IsIECCheckEnabled false, SetENOAutomatically false, UDAEnableTagReadback false
BEGIN

REGION Network 1
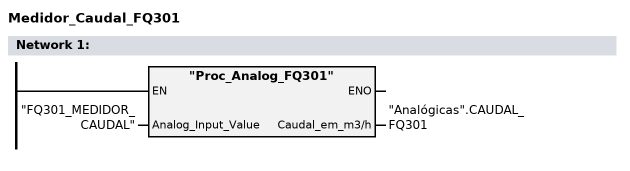
   RUNG wire#powerrail
      "Proc_Analog_FQ301"(Analog_Input_Value := "FQ301_MEDIDOR_CAUDAL", "Caudal_em_m3/h" => "Analógicas".CAUDAL_FQ301)
   END_RUNG
   // the same network as SCL:
   "Proc_Analog_FQ301"(Analog_Input_Value := "FQ301_MEDIDOR_CAUDAL",
                       "Caudal_em_m3/h" => "Analógicas".CAUDAL_FQ301);
END_REGION
END_FUNCTION

FUNCTION "Proc_Analog_FQ301" : Void   // FC12, LAD
{ S7_Optimized_Access := 'TRUE' }
VERSION : 0.1
// stored: AutoNumber true, IsIECCheckEnabled false, SetENOAutomatically false, UDAEnableTagReadback false
   VAR_INPUT
      Analog_Input_Value : Int;
   END_VAR
   VAR_OUTPUT
      "Caudal_em_m3/h" : Real;
   END_VAR
   VAR_TEMP
      "Caudal_em_%" : Real;
   END_VAR
BEGIN

REGION Network 1
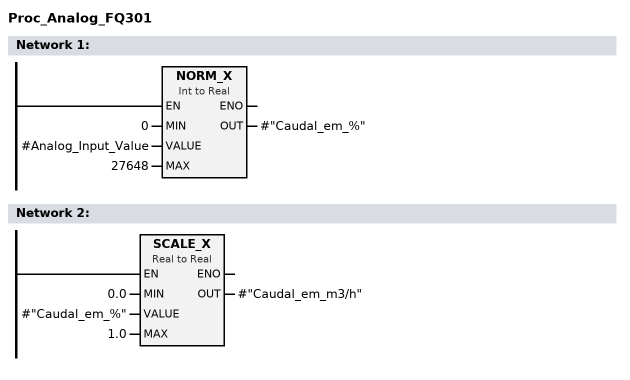
   RUNG wire#powerrail
      { S7_Templates := "[SrcType := Int, DestType := Real]"; S7_GenerateENO := "TRUE" } Normalize(min := 0, value := #Analog_Input_Value, max := 27648, out => #"Caudal_em_%")
   END_RUNG
   // the same network as SCL:
   #"Caudal_em_%" := NORM_X(MIN := 0, VALUE := #Analog_Input_Value, MAX := 27648);
END_REGION

REGION Network 2
   RUNG wire#powerrail
      { S7_Templates := "[SrcType := Real, DestType := Real]"; S7_GenerateENO := "TRUE" } Scale(min := 0.0, value := #"Caudal_em_%", max := 1.0, out => #"Caudal_em_m3/h")
   END_RUNG
   // the same network as SCL:
   #"Caudal_em_m3/h" := SCALE_X(MIN := 0.0, VALUE := #"Caudal_em_%", MAX := 1.0);
END_REGION
END_FUNCTION

FUNCTION "Sensor_Pressão_PC401" : Void   // FC13, LAD
{ S7_Optimized_Access := 'TRUE' }
VERSION : 0.1
// stored: AutoNumber true, IsIECCheckEnabled false, SetENOAutomatically false, UDAEnableTagReadback false
BEGIN

REGION Network 1
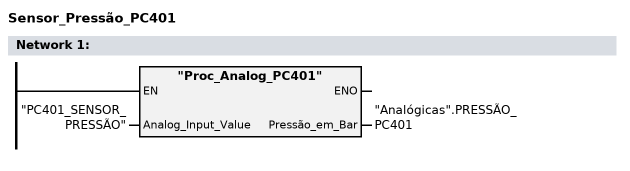
   RUNG wire#powerrail
      "Proc_Analog_PC401"(Analog_Input_Value := "PC401_SENSOR_PRESSÃO", Pressão_em_Bar => "Analógicas".PRESSÃO_PC401)
   END_RUNG
   // the same network as SCL:
   "Proc_Analog_PC401"(Analog_Input_Value := "PC401_SENSOR_PRESSÃO",
                       Pressão_em_Bar => "Analógicas".PRESSÃO_PC401);
END_REGION
END_FUNCTION

FUNCTION "Proc_Analog_PC401" : Void   // FC14, LAD
{ S7_Optimized_Access := 'TRUE' }
VERSION : 0.1
// stored: AutoNumber true, IsIECCheckEnabled false, SetENOAutomatically false, UDAEnableTagReadback false
   VAR_INPUT
      Analog_Input_Value : Int;
   END_VAR
   VAR_OUTPUT
      Pressão_em_Bar : Real;
   END_VAR
   VAR_TEMP
      "Pressão_em_%" : Real;
   END_VAR
BEGIN

REGION Network 1
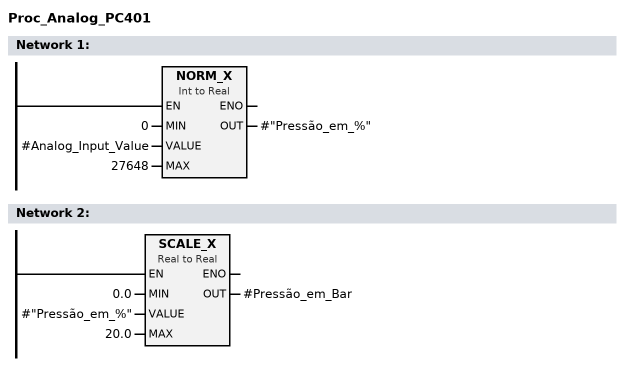
   RUNG wire#powerrail
      { S7_Templates := "[SrcType := Int, DestType := Real]"; S7_GenerateENO := "TRUE" } Normalize(min := 0, value := #Analog_Input_Value, max := 27648, out => #"Pressão_em_%")
   END_RUNG
   // the same network as SCL:
   #"Pressão_em_%" := NORM_X(MIN := 0, VALUE := #Analog_Input_Value, MAX := 27648);
END_REGION

REGION Network 2
   RUNG wire#powerrail
      { S7_Templates := "[SrcType := Real, DestType := Real]"; S7_GenerateENO := "TRUE" } Scale(min := 0.0, value := #"Pressão_em_%", max := 20.0, out => #Pressão_em_Bar)
   END_RUNG
   // the same network as SCL:
   #Pressão_em_Bar := SCALE_X(MIN := 0.0, VALUE := #"Pressão_em_%", MAX := 20.0);
END_REGION
END_FUNCTION

FUNCTION "Comando_Nível_TK02" : Void   // FC7, LAD
{ S7_Optimized_Access := 'TRUE' }
VERSION : 0.1
// stored: AutoNumber true, IsIECCheckEnabled false, SetENOAutomatically false, UDAEnableTagReadback false
   VAR_INPUT
      Nível_em_Metros : Real;
   END_VAR
   VAR_OUTPUT
      LSH : Bool;
      LSM : Bool;
      LSL : Bool;
   END_VAR
BEGIN

REGION Network 1
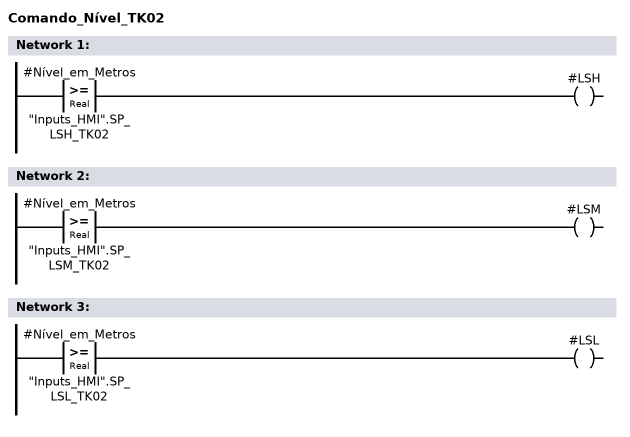
   RUNG wire#powerrail
      { S7_Templates := "SrcType := Real" } GE_Contact(in1 := #Nível_em_Metros, in2 := "Inputs_HMI".SP_LSH_TK02)
      Coil( #LSH )
   END_RUNG
   // the same network as SCL:
   #LSH := #Nível_em_Metros >= "Inputs_HMI".SP_LSH_TK02;
END_REGION

REGION Network 2
   RUNG wire#powerrail
      { S7_Templates := "SrcType := Real" } GE_Contact(in1 := #Nível_em_Metros, in2 := "Inputs_HMI".SP_LSM_TK02)
      Coil( #LSM )
   END_RUNG
   // the same network as SCL:
   #LSM := #Nível_em_Metros >= "Inputs_HMI".SP_LSM_TK02;
END_REGION

REGION Network 3
   RUNG wire#powerrail
      { S7_Templates := "SrcType := Real" } GE_Contact(in1 := #Nível_em_Metros, in2 := "Inputs_HMI".SP_LSL_TK02)
      Coil( #LSL )
   END_RUNG
   // the same network as SCL:
   #LSL := #Nível_em_Metros >= "Inputs_HMI".SP_LSL_TK02;
END_REGION
END_FUNCTION

FUNCTION "Comando_Nível_TK03" : Void   // FC10, LAD
{ S7_Optimized_Access := 'TRUE' }
VERSION : 0.1
// stored: AutoNumber true, IsIECCheckEnabled false, SetENOAutomatically false, UDAEnableTagReadback false
   VAR_INPUT
      Nível_em_Metros : Real;
   END_VAR
   VAR_OUTPUT
      LSH : Bool;
      LSM : Bool;
      LSL : Bool;
   END_VAR
BEGIN

REGION Network 1
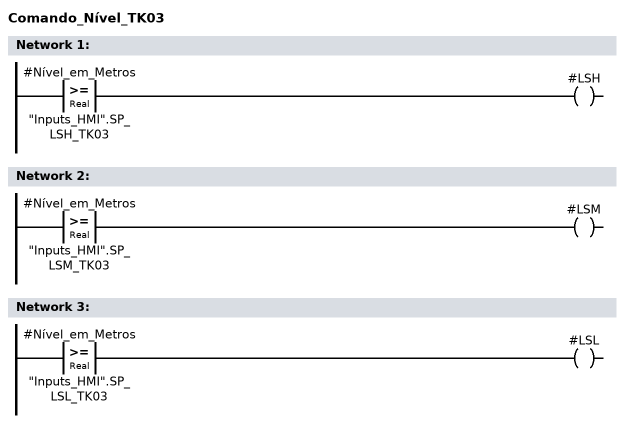
   RUNG wire#powerrail
      { S7_Templates := "SrcType := Real" } GE_Contact(in1 := #Nível_em_Metros, in2 := "Inputs_HMI".SP_LSH_TK03)
      Coil( #LSH )
   END_RUNG
   // the same network as SCL:
   #LSH := #Nível_em_Metros >= "Inputs_HMI".SP_LSH_TK03;
END_REGION

REGION Network 2
   RUNG wire#powerrail
      { S7_Templates := "SrcType := Real" } GE_Contact(in1 := #Nível_em_Metros, in2 := "Inputs_HMI".SP_LSM_TK03)
      Coil( #LSM )
   END_RUNG
   // the same network as SCL:
   #LSM := #Nível_em_Metros >= "Inputs_HMI".SP_LSM_TK03;
END_REGION

REGION Network 3
   RUNG wire#powerrail
      { S7_Templates := "SrcType := Real" } GE_Contact(in1 := #Nível_em_Metros, in2 := "Inputs_HMI".SP_LSL_TK03)
      Coil( #LSL )
   END_RUNG
   // the same network as SCL:
   #LSL := #Nível_em_Metros >= "Inputs_HMI".SP_LSL_TK03;
END_REGION
END_FUNCTION

FUNCTION "Níveis_TK02" : Void   // FC5, LAD
{ S7_Optimized_Access := 'TRUE' }
VERSION : 0.1
// stored: AutoNumber true, IsIECCheckEnabled false, SetENOAutomatically false, UDAEnableTagReadback false
BEGIN

REGION Network 1
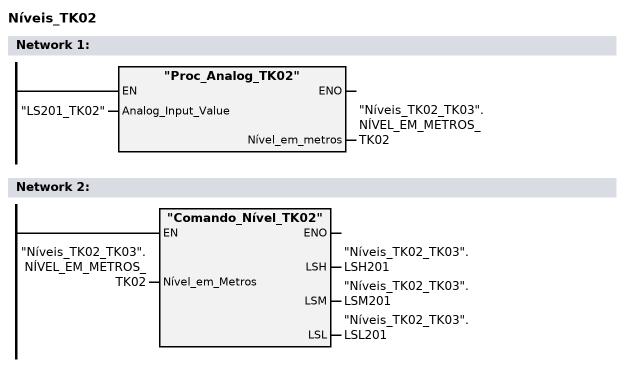
   RUNG wire#powerrail
      "Proc_Analog_TK02"(Analog_Input_Value := "LS201_TK02", Nível_em_metros => "Níveis_TK02_TK03".NÍVEL_EM_METROS_TK02)
   END_RUNG
   // the same network as SCL:
   "Proc_Analog_TK02"(Analog_Input_Value := "LS201_TK02",
                      Nível_em_metros => "Níveis_TK02_TK03".NÍVEL_EM_METROS_TK02);
END_REGION

REGION Network 2
   RUNG wire#powerrail
      "Comando_Nível_TK02"(Nível_em_Metros := "Níveis_TK02_TK03".NÍVEL_EM_METROS_TK02, LSH => "Níveis_TK02_TK03".LSH201, LSM => "Níveis_TK02_TK03".LSM201, LSL => "Níveis_TK02_TK03".LSL201)
   END_RUNG
   // the same network as SCL:
   "Comando_Nível_TK02"(Nível_em_Metros := "Níveis_TK02_TK03".NÍVEL_EM_METROS_TK02,
                        LSH => "Níveis_TK02_TK03".LSH201,
                        LSM => "Níveis_TK02_TK03".LSM201,
                        LSL => "Níveis_TK02_TK03".LSL201);
END_REGION
END_FUNCTION

FUNCTION "Proc_Analog_TK02" : Void   // FC6, LAD
{ S7_Optimized_Access := 'TRUE' }
VERSION : 0.1
// stored: AutoNumber true, IsIECCheckEnabled false, SetENOAutomatically false, UDAEnableTagReadback false
   VAR_INPUT
      Analog_Input_Value : Int;
   END_VAR
   VAR_OUTPUT
      Nível_em_metros : Real;
   END_VAR
   VAR_TEMP
      "Nível_em_%" : Real;
   END_VAR
BEGIN

REGION Network 1
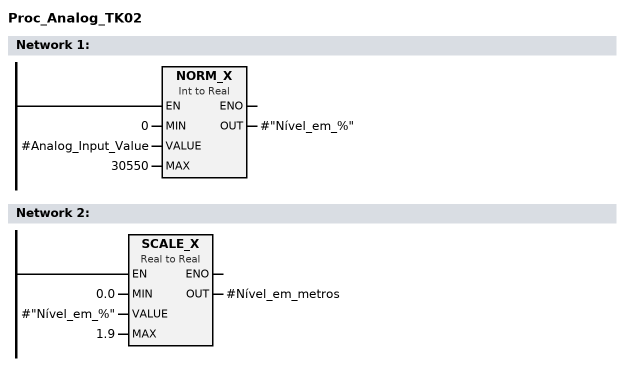
   RUNG wire#powerrail
      { S7_Templates := "[SrcType := Int, DestType := Real]"; S7_GenerateENO := "TRUE" } Normalize(min := 0, value := #Analog_Input_Value, max := 30550, out => #"Nível_em_%")
   END_RUNG
   // the same network as SCL:
   #"Nível_em_%" := NORM_X(MIN := 0, VALUE := #Analog_Input_Value, MAX := 30550);
END_REGION

REGION Network 2
   RUNG wire#powerrail
      { S7_Templates := "[SrcType := Real, DestType := Real]"; S7_GenerateENO := "TRUE" } Scale(min := 0.0, value := #"Nível_em_%", max := 1.9, out => #Nível_em_metros)
   END_RUNG
   // the same network as SCL:
   #Nível_em_metros := SCALE_X(MIN := 0.0, VALUE := #"Nível_em_%", MAX := 1.9);
END_REGION
END_FUNCTION

FUNCTION "Níveis_TK03" : Void   // FC8, LAD
{ S7_Optimized_Access := 'TRUE' }
VERSION : 0.1
// stored: AutoNumber true, IsIECCheckEnabled false, SetENOAutomatically false, UDAEnableTagReadback false
BEGIN

REGION Network 1
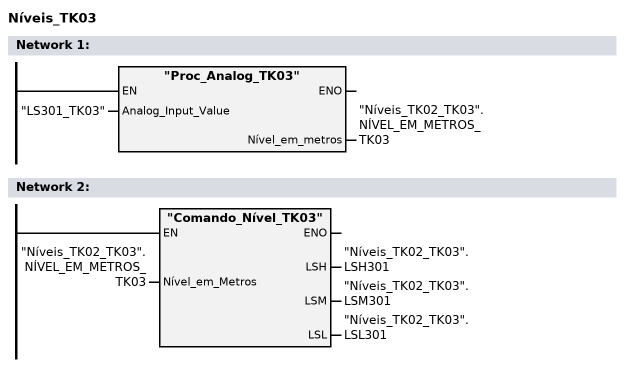
   RUNG wire#powerrail
      "Proc_Analog_TK03"(Analog_Input_Value := "LS301_TK03", Nível_em_metros => "Níveis_TK02_TK03".NÍVEL_EM_METROS_TK03)
   END_RUNG
   // the same network as SCL:
   "Proc_Analog_TK03"(Analog_Input_Value := "LS301_TK03",
                      Nível_em_metros => "Níveis_TK02_TK03".NÍVEL_EM_METROS_TK03);
END_REGION

REGION Network 2
   RUNG wire#powerrail
      "Comando_Nível_TK03"(Nível_em_Metros := "Níveis_TK02_TK03".NÍVEL_EM_METROS_TK03, LSH => "Níveis_TK02_TK03".LSH301, LSM => "Níveis_TK02_TK03".LSM301, LSL => "Níveis_TK02_TK03".LSL301)
   END_RUNG
   // the same network as SCL:
   "Comando_Nível_TK03"(Nível_em_Metros := "Níveis_TK02_TK03".NÍVEL_EM_METROS_TK03,
                        LSH => "Níveis_TK02_TK03".LSH301,
                        LSM => "Níveis_TK02_TK03".LSM301,
                        LSL => "Níveis_TK02_TK03".LSL301);
END_REGION
END_FUNCTION

FUNCTION "Proc_Analog_TK03" : Void   // FC9, LAD
{ S7_Optimized_Access := 'TRUE' }
VERSION : 0.1
// stored: AutoNumber true, IsIECCheckEnabled false, SetENOAutomatically false, UDAEnableTagReadback false
   VAR_INPUT
      Analog_Input_Value : Int;
   END_VAR
   VAR_OUTPUT
      Nível_em_metros : Real;
   END_VAR
   VAR_TEMP
      "Nível_em_%" : Real;
   END_VAR
BEGIN

REGION Network 1
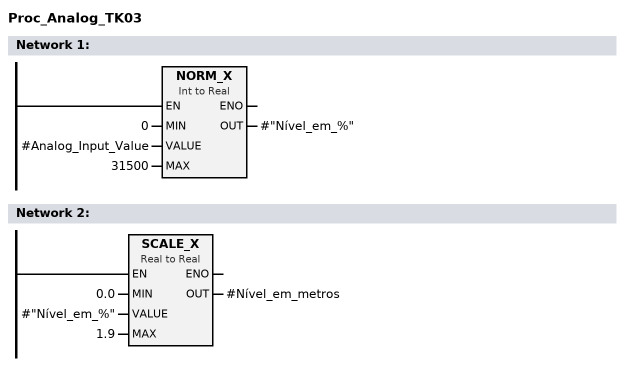
   RUNG wire#powerrail
      { S7_Templates := "[SrcType := Int, DestType := Real]"; S7_GenerateENO := "TRUE" } Normalize(min := 0, value := #Analog_Input_Value, max := 31500, out => #"Nível_em_%")
   END_RUNG
   // the same network as SCL:
   #"Nível_em_%" := NORM_X(MIN := 0, VALUE := #Analog_Input_Value, MAX := 31500);
END_REGION

REGION Network 2
   RUNG wire#powerrail
      { S7_Templates := "[SrcType := Real, DestType := Real]"; S7_GenerateENO := "TRUE" } Scale(min := 0.0, value := #"Nível_em_%", max := 1.9, out => #Nível_em_metros)
   END_RUNG
   // the same network as SCL:
   #Nível_em_metros := SCALE_X(MIN := 0.0, VALUE := #"Nível_em_%", MAX := 1.9);
END_REGION
END_FUNCTION

FUNCTION "Alim_Processo" : Void   // FC1, LAD
{ S7_Optimized_Access := 'TRUE' }
VERSION : 0.1
// stored: AutoNumber true, IsIECCheckEnabled false, SetENOAutomatically false, UDAEnableTagReadback false
BEGIN

REGION Network 1: Etapa 10 (INÍCIO)
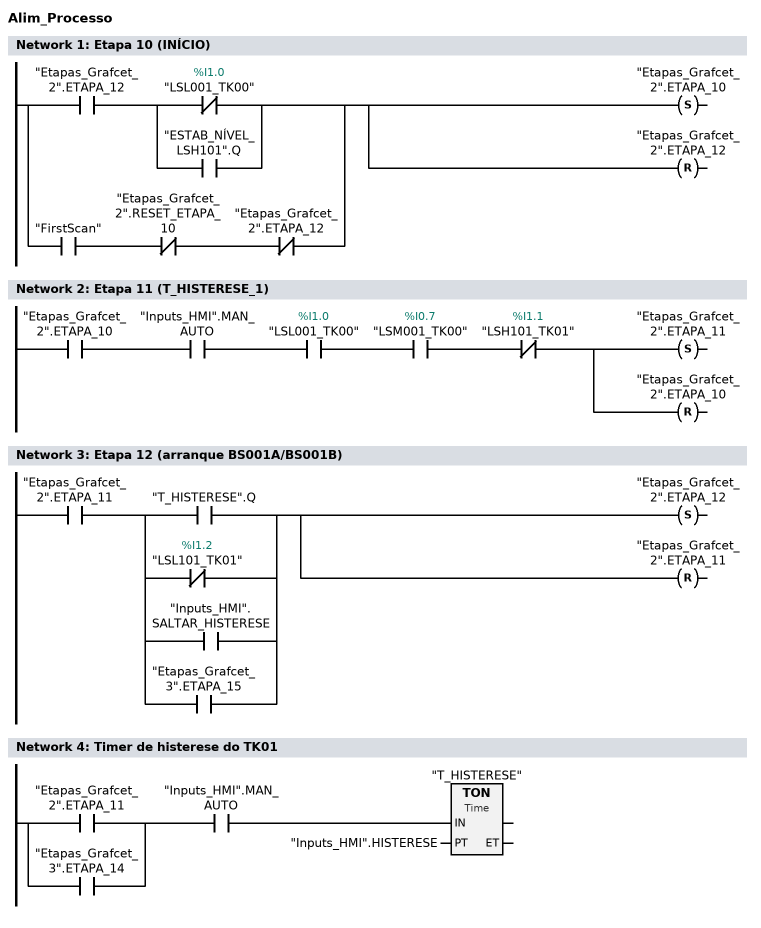
   RUNG wire#powerrail
      Contact( "Etapas_Grafcet_2".ETAPA_12 )
      wire#w1
      I_Contact( "LSL001_TK00" )
      wire#w2
      S_Coil( "Etapas_Grafcet_2".ETAPA_10 )
   END_RUNG
   RUNG wire#w1
      Contact( "ESTAB_NÍVEL_LSH101".Q )
   END_RUNG wire#w2
   RUNG wire#powerrail
      Contact( "FirstScan" )
      I_Contact( "Etapas_Grafcet_2".RESET_ETAPA_10 )
      I_Contact( "Etapas_Grafcet_2".ETAPA_12 )
   END_RUNG wire#w2
   RUNG wire#w2
      R_Coil( "Etapas_Grafcet_2".ETAPA_12 )
   END_RUNG
   // the same network as SCL:
   IF ("Etapas_Grafcet_2".ETAPA_12 AND (NOT "LSL001_TK00" OR "ESTAB_NÍVEL_LSH101".Q)) OR ("FirstScan" AND NOT "Etapas_Grafcet_2".RESET_ETAPA_10 AND NOT "Etapas_Grafcet_2".ETAPA_12) THEN
       "Etapas_Grafcet_2".ETAPA_10 := TRUE;
       "Etapas_Grafcet_2".ETAPA_12 := FALSE;
   END_IF;
END_REGION

REGION Network 2: Etapa 11 (T_HISTERESE_1)
   RUNG wire#powerrail
      Contact( "Etapas_Grafcet_2".ETAPA_10 )
      Contact( "Inputs_HMI".MAN_AUTO )
      Contact( "LSL001_TK00" )
      Contact( "LSM001_TK00" )
      I_Contact( "LSH101_TK01" )
      wire#w1
      S_Coil( "Etapas_Grafcet_2".ETAPA_11 )
   END_RUNG
   RUNG wire#w1
      R_Coil( "Etapas_Grafcet_2".ETAPA_10 )
   END_RUNG
   // the same network as SCL:
   IF "Etapas_Grafcet_2".ETAPA_10 AND "Inputs_HMI".MAN_AUTO AND "LSL001_TK00" AND "LSM001_TK00" AND NOT "LSH101_TK01" THEN
       "Etapas_Grafcet_2".ETAPA_11 := TRUE;
       "Etapas_Grafcet_2".ETAPA_10 := FALSE;
   END_IF;
END_REGION

REGION Network 3: Etapa 12 (arranque BS001A/BS001B)
   RUNG wire#powerrail
      Contact( "Etapas_Grafcet_2".ETAPA_11 )
      wire#w1
      Contact( "T_HISTERESE".Q )
      wire#w2
      S_Coil( "Etapas_Grafcet_2".ETAPA_12 )
   END_RUNG
   RUNG wire#w1
      I_Contact( "LSL101_TK01" )
   END_RUNG wire#w2
   RUNG wire#w1
      Contact( "Inputs_HMI".SALTAR_HISTERESE )
   END_RUNG wire#w2
   RUNG wire#w1
      Contact( "Etapas_Grafcet_3".ETAPA_15 )
   END_RUNG wire#w2
   RUNG wire#w2
      R_Coil( "Etapas_Grafcet_2".ETAPA_11 )
   END_RUNG
   // the same network as SCL:
   IF "Etapas_Grafcet_2".ETAPA_11 AND ("T_HISTERESE".Q OR NOT "LSL101_TK01" OR "Inputs_HMI".SALTAR_HISTERESE OR "Etapas_Grafcet_3".ETAPA_15) THEN
       "Etapas_Grafcet_2".ETAPA_12 := TRUE;
       "Etapas_Grafcet_2".ETAPA_11 := FALSE;
   END_IF;
END_REGION

REGION Network 4: Timer de histerese do TK01
   RUNG wire#powerrail
      Contact( "Etapas_Grafcet_2".ETAPA_11 )
      wire#w1
      Contact( "Inputs_HMI".MAN_AUTO )
      { S7_Templates := "time_type := Time" } "T_HISTERESE".TON(pt := "Inputs_HMI".HISTERESE, et =>)
   END_RUNG
   RUNG wire#powerrail
      Contact( "Etapas_Grafcet_3".ETAPA_14 )
   END_RUNG wire#w1
   // the same network as SCL:
   "T_HISTERESE".TON(IN := ("Etapas_Grafcet_2".ETAPA_11 OR "Etapas_Grafcet_3".ETAPA_14) AND "Inputs_HMI".MAN_AUTO,
                     PT := "Inputs_HMI".HISTERESE);
END_REGION
END_FUNCTION

FUNCTION "Ciclo_Tratamento" : Void   // FC4, LAD
{ S7_Optimized_Access := 'TRUE' }
VERSION : 0.1
// stored: AutoNumber true, IsIECCheckEnabled false, SetENOAutomatically false, UDAEnableTagReadback false
   VAR_TEMP   // added for the SCL form of the ladder/FBD networks
      _w1 : Bool;
      _w2 : Bool;
   END_VAR
BEGIN

REGION Network 1: Etapa 1 (INÍCIO)
